Fanuc KAREL source: kd00004.KL

-- PROVISIONAL review KL for V1013-1; original PC SHA256 357ad229c04065b93161180d755f1119893f9ca71272e7da16a1d974bff7769d
-- Incomplete behavior may be omitted. Consult companion uncertainty JSON. Do not deploy.
PROGRAM KD00004
%NOLOCKGROUP
VAR
  I : INTEGER
  J : INTEGER
  B : BOOLEAN
  R : REAL
  S : STRING[80]
BEGIN
  -- UNRESOLVED_PC offsets 5-12; opcodes 9D,23
  -- UNRESOLVED_PC offsets 17-21; opcodes 7F
END KD00004
